TYPE (* a Struct holding 2 Object IDs *)
  (* Version 1.0, 2026-05-28, Franz Höpfinger, Demmler Andreas Fahrzeugbau *)
  PACKAGE isobus::UT::Q::types;
  IMPORT isobus::UT::Q::const::IDs::ID_NULL;
  s2ObjectIDs : STRUCT
    u16ObjId : UINT := ID_NULL; (* Object ID Softkey *)
    u16ObjIdA : UINT := ID_NULL; (* Object ID AUX *)
  END_STRUCT;
END_TYPE
